// TwinCAT 3 PLC project Nepionic_Log_OTel
// Title: Nepionic_Log_OTel
// Company: Nepionic
// Author: Nepionic
// ProjectVersion: 0.1.0
// ProgramVersion: 3.1.4026.22
// libraries:
//   [Nepionic_Log], * (Nepionic)
//   Tc2_System, * (Beckhoff Automation GmbH)
//   Tc2_Utilities, * (Beckhoff Automation GmbH)
// project tree:
//   Lib/ OTelLogAppender.TcPOU, OTelLogEntry.TcDUT (not stored), OTelLogRing.TcDUT (not stored)

// ---- Lib/OTelLogAppender.TcPOU
{attribute 'linkalways'}
{attribute 'no_explicit_call' := 'This FB is a CLASS and must be accessed using methods or properties'}
{attribute 'enable_dynamic_creation'}
// DEPRECATED: superseded by Nepionic_Log_Klein.KleinEventAppender, which writes the
// same proven seqlock ring-buffer wire shape into a KleinEventEntry/KleinEventRing pair
// consumed by the Klein collector's ADS receiver (github.com/siyka-au/klein,
// internal/receiver/ads/eventring.go) instead of otelcol-ads. New projects should
// reference Nepionic_Log_Klein instead of Nepionic_Log_OTel. This library is kept for
// existing consumers and is not scheduled for removal.
/// OTel log appender for Nepionic_Log.
/// Implements `LogAppender` by writing structured log entries directly into its
/// own `OTelLogRing` field (`Ring`), which is exposed as an ADS symbol and
/// consumed by the Go `otelcol-ads` collector.
///
/// The ring is owned by the appender — no external ring declaration is needed.
/// Just declare the appender in a PROGRAM or GVL so TwinCAT generates an ADS
/// symbol for it, then point the collector at `<PROGRAM>.<var_name>.Ring`.
///
/// Usage:
/// ```st
/// // startup (e.g. MAIN FB_Init)
/// GetLogManager().Register(otel_appender);
///
/// // otelcol-ads config:
/// //   symbol: MAIN.otel_appender.Ring
/// ```
FUNCTION_BLOCK PUBLIC OTelLogAppender IMPLEMENTS Nepionic_Log.LogAppender
VAR
	{attribute 'otelcol_role' := 'log_ring'}
	ring : OTelLogRing;
	_level : Nepionic_Log.LogLevel := Nepionic_Log.LogLevel.Debug;
END_VAR

METHOD PUBLIC Append : BOOL
VAR_INPUT
	level : Nepionic_Log.LogLevel;
	message : Tc2_System.T_MaxString;
	source : Tc2_System.T_MaxString;
	attributes : ARRAY[0..9] OF Nepionic_Log.LogAttribute;
	attribute_count : USINT;
END_VAR
VAR
	slot_idx : UDINT;
	expected_gen : UDINT;
	file_time : ULINT;
	i : USINT;
END_VAR
slot_idx := ring.head MOD ring.capacity;
expected_gen := (ring.head / ring.capacity + 1) * 2;

// Mark slot as being written (ODD sequence = write in progress)
ring.entries[slot_idx].sequence := expected_gen - 1;

// Timestamp — Windows FILETIME → Unix nanoseconds
file_time := Tc2_Utilities.F_GetSystemTime();
ring.entries[slot_idx].timestamp := (file_time - 116444736000000000) * 100;

// Severity mapping
CASE level OF
	Nepionic_Log.LogLevel.Debug:
		ring.entries[slot_idx].severity := 0;
	Nepionic_Log.LogLevel.Information:
		ring.entries[slot_idx].severity := 1;
	Nepionic_Log.LogLevel.Warning:
		ring.entries[slot_idx].severity := 2;
	Nepionic_Log.LogLevel.Error:
		ring.entries[slot_idx].severity := 3;
	Nepionic_Log.LogLevel.Fatal:
		ring.entries[slot_idx].severity := 4;
ELSE
	ring.entries[slot_idx].severity := 1;
END_CASE

// Payload
ring.entries[slot_idx].message := message;
ring.entries[slot_idx].source := source;
ring.entries[slot_idx].attribute_count := USINT_TO_UDINT(attribute_count);
FOR i := 0 TO 9 DO
	ring.entries[slot_idx].attributes[i] := attributes[i];
END_FOR

// Commit slot (EVEN sequence = ready for reader)
ring.entries[slot_idx].sequence := expected_gen;

// Increment overflow counter each time the write pointer wraps back to slot 0.
IF slot_idx = 0 AND ring.head > 0 THEN
	ring.overflow_cnt := ring.overflow_cnt + 1;
END_IF

// Advance write cursor
ring.head := ring.head + 1;

Append := TRUE;
END_METHOD

{attribute 'monitoring' := 'call'}
PROPERTY PUBLIC Level : Nepionic_Log.LogLevel
GET // PUBLIC
Level := _level;
END_GET
SET // PUBLIC
_level := Level;
END_SET
END_PROPERTY

END_FUNCTION_BLOCK
